//==================================================================================================
//							Beckhoff Automation Poland
//									23.05.2017
// 	v1.0	|| TC v 3.1.4020.32		|| - pierwsza wersja
//==================================================================================================
{attribute 'qualified_only'}
VAR_GLOBAL PERSISTENT
	arrEvent								: ARRAY [1..GVL_EHS.diNoOfEvents] OF ST_EventHistoricalSimplePersistent;
END_VAR

(* stored: Version 1.1.0.1, ProductVersion 3.1.4022.6
   GVL GVL_EHSP: Id {7b42e079-7bfd-4d59-811a-19d7abc08160} *)
